   cmCathodeMainPnP2AxisZ.commandConfiguration.moveVelocity.velocity := 0.0;
   cmCathodeMainPnP2AxisZ.commandConfiguration.moveVelocity.acceleration := -1.0;
   cmCathodeMainPnP2AxisZ.commandConfiguration.moveVelocity.deceleration := -1.0;
   cmCathodeMainPnP2AxisZ.commandConfiguration.moveVelocity.jerk := -1.0;
   cmCathodeMainPnP2AxisZ.commandConfiguration.moveVelocity.direction := 0;
   cmCathodeMainPnP2AxisZ.commandConfiguration.moveVelocity.positionControlled := TRUE;
   cmCathodeMainPnP2AxisZ.commandConfiguration.moveVelocity.velocityChangeOnTheFly := FALSE;
   cmCathodeMainPnP2AxisZ.commandConfiguration.stop.deceleration := -1.0;
   cmCathodeMainPnP2AxisZ.commandConfiguration.stop.jerk := -1.0;
   cmCathodeMainPnP2AxisZ.commandConfiguration.stop.abortAcceleration := FALSE;
   cmCathodeMainPnP2AxisZ.commandConfiguration.fastStop.deceleration := -1.0;
   cmCathodeMainPnP2AxisZ.commandConfiguration.fastStop.jerk := -1.0;
   cmCathodeMainPnP2AxisZ.commandConfiguration.fastStop.abortAcceleration := FALSE;
   cmCathodeMainPnP2AxisZ.commandConfiguration.fastStop.replaceStopPossible := FALSE;
   cmCathodeMainPnP2AxisZ.commandConfiguration.torqueLimiting.limit := -1.0;
   cmCathodeMainPnP2AxisZ.commandConfiguration.torqueLimiting.mode := 0;
   cmCathodeMainPnP2AxisZ.commandConfiguration.homing.position := 0.0;
   cmCathodeMainPnP2AxisZ.commandConfiguration.homing.mode := 0;
   cmCathodeMainPnP2AxisZ.commandConfiguration.homing.sensor := 0;
   cmCathodeMainPnP2AxisZ.commandConfiguration.homing.extendedMode := -1;
   cmCathodeMainPnP2AxisZ.commandConfiguration.homing.extendedModeTorqueLimit := 0.0;
   cmCathodeMainPnP2AxisZ.commandConfiguration.homing.extendedModeTargetPosition := 0.0;
   cmCathodeMainPnP2AxisZ.commandConfiguration.posRelative.distance := 0.0;
   cmCathodeMainPnP2AxisZ.commandConfiguration.posRelative.velocity := -1.0;
   cmCathodeMainPnP2AxisZ.commandConfiguration.posRelative.acceleration := -1.0;
   cmCathodeMainPnP2AxisZ.commandConfiguration.posRelative.deceleration := -1.0;
   cmCathodeMainPnP2AxisZ.commandConfiguration.posRelative.jerk := -1.0;
   cmCathodeMainPnP2AxisZ.commandConfiguration.posRelative.direction := 0;
   cmCathodeMainPnP2AxisZ.commandConfiguration.posAbsolute.position := 0.0;
   cmCathodeMainPnP2AxisZ.commandConfiguration.posAbsolute.velocity := -1.0;
   cmCathodeMainPnP2AxisZ.commandConfiguration.posAbsolute.acceleration := -1.0;
   cmCathodeMainPnP2AxisZ.commandConfiguration.posAbsolute.deceleration := -1.0;
   cmCathodeMainPnP2AxisZ.commandConfiguration.posAbsolute.jerk := -1.0;
   cmCathodeMainPnP2AxisZ.commandConfiguration.posAbsolute.direction := 1;
   cmCathodeMainPnP2AxisZ.commandConfiguration.posAbsolute.positionChangeOnTheFly := FALSE;
   cmCathodeMainPnP2AxisZ.commandConfiguration.posAbsolute.velocityChangeOnTheFly := FALSE;
   cmCathodeMainPnP2AxisZ.commandConfiguration.posSuperimposed.distance := 0.0;
   cmCathodeMainPnP2AxisZ.commandConfiguration.posSuperimposed.velocityDiff := -1.0;
   cmCathodeMainPnP2AxisZ.commandConfiguration.posSuperimposed.acceleration := -1.0;
   cmCathodeMainPnP2AxisZ.commandConfiguration.posSuperimposed.deceleration := -1.0;
   cmCathodeMainPnP2AxisZ.commandConfiguration.posSuperimposed.jerk := -1.0;
   cmCathodeMainPnP2AxisZ.commandConfiguration.posSuperimposed.direction := 0;
   cmCathodeMainPnP2AxisZ.commandConfiguration.haltSuperimposed.deceleration := -1.0;
   cmCathodeMainPnP2AxisZ.commandConfiguration.haltSuperimposed.jerk := -1.0;
   cmCathodeMainPnP2AxisZ.commandConfiguration.haltSuperimposed.abortAcceleration := FALSE;
   cmCathodeMainPnP2AxisZ.commandConfiguration.gearInRelative.ratioNumerator := 1;
   cmCathodeMainPnP2AxisZ.commandConfiguration.gearInRelative.ratioDenominator := 1;
   cmCathodeMainPnP2AxisZ.commandConfiguration.gearInRelative.acceleration := -1.0;
   cmCathodeMainPnP2AxisZ.commandConfiguration.gearInRelative.deceleration := -1.0;
   cmCathodeMainPnP2AxisZ.commandConfiguration.gearInRelative.jerk := -1.0;
   cmCathodeMainPnP2AxisZ.commandConfiguration.gearInRelative.ratioChangeOnTheFly := FALSE;
   cmCathodeMainPnP2AxisZ.commandConfiguration.gearInAbsolute.ratioNumerator := 1;
   cmCathodeMainPnP2AxisZ.commandConfiguration.gearInAbsolute.ratioDenominator := 1;
   cmCathodeMainPnP2AxisZ.commandConfiguration.gearInAbsolute.masterSyncPosition := 0.0;
   cmCathodeMainPnP2AxisZ.commandConfiguration.gearInAbsolute.slaveSyncPosition := 0.0;
   cmCathodeMainPnP2AxisZ.commandConfiguration.gearInAbsolute.syncProfileReference := 1;
   cmCathodeMainPnP2AxisZ.commandConfiguration.gearInAbsolute.masterStartDistance := 0.0;
   cmCathodeMainPnP2AxisZ.commandConfiguration.gearInAbsolute.velocity := -1.0;
   cmCathodeMainPnP2AxisZ.commandConfiguration.gearInAbsolute.acceleration := -1.0;
   cmCathodeMainPnP2AxisZ.commandConfiguration.gearInAbsolute.deceleration := -1.0;
   cmCathodeMainPnP2AxisZ.commandConfiguration.gearInAbsolute.jerk := -1.0;
   cmCathodeMainPnP2AxisZ.commandConfiguration.gearInAbsolute.syncDirection := 1;
   cmCathodeMainPnP2AxisZ.commandConfiguration.gearInAbsolute.ratioChangeOnTheFly := FALSE;
   cmCathodeMainPnP2AxisZ.commandConfiguration.gearInVelocity.continuousUpdate := FALSE;
   cmCathodeMainPnP2AxisZ.commandConfiguration.gearInVelocity.ratioNumerator := 1;
   cmCathodeMainPnP2AxisZ.commandConfiguration.gearInVelocity.ratioDenominator := 1;
   cmCathodeMainPnP2AxisZ.commandConfiguration.gearInVelocity.acceleration := -1.0;
   cmCathodeMainPnP2AxisZ.commandConfiguration.gearInVelocity.deceleration := -1.0;
   cmCathodeMainPnP2AxisZ.commandConfiguration.gearInVelocity.jerk := -1.0;
   cmCathodeMainPnP2AxisZ.commandConfiguration.gearInVelocity.positionControlled := FALSE;
   cmCathodeMainPnP2AxisZ.commandConfiguration.camIn.masterOffset := 0.0;
   cmCathodeMainPnP2AxisZ.commandConfiguration.camIn.slaveOffset := 0.0;
   cmCathodeMainPnP2AxisZ.commandConfiguration.camIn.masterScaling := 1.0;
   cmCathodeMainPnP2AxisZ.commandConfiguration.camIn.slaveScaling := 1.0;
   cmCathodeMainPnP2AxisZ.commandConfiguration.camIn.masterSyncPosition := 0.0;
   cmCathodeMainPnP2AxisZ.commandConfiguration.camIn.syncProfileReference := 1;
   cmCathodeMainPnP2AxisZ.commandConfiguration.camIn.masterStartDistance := 0.0;
   cmCathodeMainPnP2AxisZ.commandConfiguration.camIn.velocity := -1.0;
   cmCathodeMainPnP2AxisZ.commandConfiguration.camIn.acceleration := -1.0;
   cmCathodeMainPnP2AxisZ.commandConfiguration.camIn.deceleration := -1.0;
   cmCathodeMainPnP2AxisZ.commandConfiguration.camIn.jerk := -1.0;
   cmCathodeMainPnP2AxisZ.commandConfiguration.camIn.applicationMode := 0;
   cmCathodeMainPnP2AxisZ.commandConfiguration.camIn.syncDirection := 1;
   cmCathodeMainPnP2AxisZ.commandConfiguration.gearOutCamOut.slavePosition := 0.0;
   cmCathodeMainPnP2AxisZ.commandConfiguration.gearOutCamOut.syncProfileReference := 1;
   cmCathodeMainPnP2AxisZ.commandConfiguration.gearOutCamOut.masterStopDistance := 0.0;
   cmCathodeMainPnP2AxisZ.commandConfiguration.gearOutCamOut.deceleration := -1.0;
   cmCathodeMainPnP2AxisZ.commandConfiguration.gearOutCamOut.jerk := -1.0;
   cmCathodeMainPnP2AxisZ.commandConfiguration.gearOutCamOut.syncOutDirection := 3;
   cmCathodeMainPnP2AxisZ.commandConfiguration.gearOutCamOut.gearOutCamOutMode := -1;
   cmCathodeMainPnP2AxisZ.commandConfiguration.phasing.phaseShift := 0.0;
   cmCathodeMainPnP2AxisZ.commandConfiguration.phasing.velocity := -1.0;
   cmCathodeMainPnP2AxisZ.commandConfiguration.phasing.acceleration := -1.0;
   cmCathodeMainPnP2AxisZ.commandConfiguration.phasing.deceleration := -1.0;
   cmCathodeMainPnP2AxisZ.commandConfiguration.phasing.jerk := -1.0;
   cmCathodeMainPnP2AxisZ.commandConfiguration.phasing.profileReference := 0;
   cmCathodeMainPnP2AxisZ.commandConfiguration.phasing.phasingDistance := 0.0;
   cmCathodeMainPnP2AxisZ.commandConfiguration.phasing.startPosition := 0.0;
   cmCathodeMainPnP2AxisZ.commandConfiguration.phasing.direction := 3;
   cmCathodeMainPnP2AxisZ.commandConfiguration.phasing.phaseAbsolute := TRUE;
   cmCathodeMainPnP2AxisZ.commandConfiguration.phasing.phaseShiftChangeOnTheFly := FALSE;
   cmCathodeMainPnP2AxisZ.commandConfiguration.offset.offset := 0.0;
   cmCathodeMainPnP2AxisZ.commandConfiguration.offset.profileReference := 1;
   cmCathodeMainPnP2AxisZ.commandConfiguration.offset.offsetDistance := 0.0;
   cmCathodeMainPnP2AxisZ.commandConfiguration.offset.startPosition := 0.0;
   cmCathodeMainPnP2AxisZ.commandConfiguration.offset.direction := 3;
   cmCathodeMainPnP2AxisZ.commandConfiguration.offset.offsetAbsolute := TRUE;
   cmCathodeMainPnP2AxisZ.commandConfiguration.offset.offsetChangeOnTheFly := FALSE;
   cmCathodeMainPnP2AxisZ.commands.enableAxis := FALSE;
   cmCathodeMainPnP2AxisZ.commands.resetAxis := FALSE;
   cmCathodeMainPnP2AxisZ.commands.openBrake := FALSE;
   cmCathodeMainPnP2AxisZ.commands.jogForward := FALSE;
   cmCathodeMainPnP2AxisZ.commands.jogBackward := FALSE;
   cmCathodeMainPnP2AxisZ.commands.moveVelocity := FALSE;
   cmCathodeMainPnP2AxisZ.commands.stop := FALSE;
   cmCathodeMainPnP2AxisZ.commands.fastStop := FALSE;
   cmCathodeMainPnP2AxisZ.commands.torqueLimiting := FALSE;
   cmCathodeMainPnP2AxisZ.commands.homing := FALSE;
   cmCathodeMainPnP2AxisZ.commands.posRelative := FALSE;
   cmCathodeMainPnP2AxisZ.commands.posAbsolute := FALSE;
   cmCathodeMainPnP2AxisZ.commands.posSuperimposed := FALSE;
   cmCathodeMainPnP2AxisZ.commands.haltSuperimposed := FALSE;
   cmCathodeMainPnP2AxisZ.commands.selectSetPosition := -1;
   cmCathodeMainPnP2AxisZ.commands.reset := FALSE;
   cmCathodeMainPnP2AxisZ.monitoring.valid := FALSE;
   cmCathodeMainPnP2AxisZ.monitoring.busy := TRUE;
   cmCathodeMainPnP2AxisZ.monitoring.error := TRUE;
   cmCathodeMainPnP2AxisZ.monitoring.status := 16#8600;
   cmCathodeMainPnP2AxisZ.monitoring.subfunctionStatus := 16#8001;
   cmCathodeMainPnP2AxisZ.monitoring.axisEnabled := FALSE;
   cmCathodeMainPnP2AxisZ.monitoring.resetActive := FALSE;
   cmCathodeMainPnP2AxisZ.monitoring.inVelocity := FALSE;
   cmCathodeMainPnP2AxisZ.monitoring.inLimitation := FALSE;
   cmCathodeMainPnP2AxisZ.monitoring.inClamping := FALSE;
   cmCathodeMainPnP2AxisZ.monitoring.startSync := FALSE;
   cmCathodeMainPnP2AxisZ.monitoring.inSync := FALSE;
   cmCathodeMainPnP2AxisZ.monitoring.inSimulation := FALSE;
   cmCathodeMainPnP2AxisZ.monitoring.jogSelected := FALSE;
   cmCathodeMainPnP2AxisZ.monitoring.moveVelocitySelected := FALSE;
   cmCathodeMainPnP2AxisZ.monitoring.stopSelected := FALSE;
   cmCathodeMainPnP2AxisZ.monitoring.fastStopSelected := FALSE;
   cmCathodeMainPnP2AxisZ.monitoring.torqueLimitingSelected := FALSE;
   cmCathodeMainPnP2AxisZ.monitoring.homingSelected := FALSE;
   cmCathodeMainPnP2AxisZ.monitoring.posRelativeSelected := FALSE;
   cmCathodeMainPnP2AxisZ.monitoring.posAbsoluteSelected := FALSE;
   cmCathodeMainPnP2AxisZ.monitoring.posSuperimposedSelected := FALSE;
   cmCathodeMainPnP2AxisZ.monitoring.haltSuperimposedSelected := FALSE;
   cmCathodeMainPnP2AxisZ.monitoring.commandBusy := FALSE;
   cmCathodeMainPnP2AxisZ.monitoring.commandDone := FALSE;
   cmCathodeMainPnP2AxisZ.monitoring.commandAborted := FALSE;
   cmCathodeMainPnP2AxisZ.monitoring.homingCommandBusy := FALSE;
   cmCathodeMainPnP2AxisZ.monitoring.homingCommandDone := FALSE;
   cmCathodeMainPnP2AxisZ.monitoring.homingCommandAborted := FALSE;
   cmCathodeMainPnP2AxisZ.monitoring.superimposedBusy := FALSE;
   cmCathodeMainPnP2AxisZ.monitoring.superimposedDone := FALSE;
   cmCathodeMainPnP2AxisZ.monitoring.superimposedAborted := FALSE;
   cmCathodeMainPnP2AxisZ.monitoring.actualPosition := 2.382;
   cmCathodeMainPnP2AxisZ.monitoring.actualSpeed := 0.0;
   cmCathodeMainPnP2AxisZ.monitoring.speedUnit := 1062;
   cmCathodeMainPnP2AxisZ.monitoring.positionUnit := 1013;
   cmCathodeMainPnP2AxisZ.monitoring.axisType := 1;
   cmCathodeMainPnP2AxisZ.monitoring.interlockGeneralOut := TRUE;
   cmCathodeMainPnP2AxisZ.monitoring.interlockJogForwardOut := TRUE;
   cmCathodeMainPnP2AxisZ.monitoring.interlockJogBackwardOut := TRUE;
   cmCathodeAlignTableAxisX.commandConfiguration.generalSettings.stopOnError := TRUE;
   cmCathodeAlignTableAxisX.commandConfiguration.generalSettings.resetWithRestart := FALSE;
   cmCathodeAlignTableAxisX.commandConfiguration.generalSettings.abortWaitingSyncCmd := TRUE;
   cmCathodeAlignTableAxisX.commandConfiguration.power.startMode := 1;
   cmCathodeAlignTableAxisX.commandConfiguration.power.stopMode := 0;
   cmCathodeAlignTableAxisX.commandConfiguration.power.syncMotionSimulation := FALSE;
   cmCathodeAlignTableAxisX.commandConfiguration.power.syncMotionSimulationExtendedMode := -1;
   cmCathodeAlignTableAxisX.commandConfiguration.jog.velocity := 0.0;
   cmCathodeAlignTableAxisX.commandConfiguration.jog.acceleration := -1.0;
   cmCathodeAlignTableAxisX.commandConfiguration.jog.deceleration := -1.0;
   cmCathodeAlignTableAxisX.commandConfiguration.jog.jerk := -1.0;
   cmCathodeAlignTableAxisX.commandConfiguration.jog.positionControlled := TRUE;
   cmCathodeAlignTableAxisX.commandConfiguration.jog.increment := 0.0;
   cmCathodeAlignTableAxisX.commandConfiguration.jog.mode := 0;
   cmCathodeAlignTableAxisX.commandConfiguration.moveVelocity.velocity := 0.0;
   cmCathodeAlignTableAxisX.commandConfiguration.moveVelocity.acceleration := -1.0;
   cmCathodeAlignTableAxisX.commandConfiguration.moveVelocity.deceleration := -1.0;
   cmCathodeAlignTableAxisX.commandConfiguration.moveVelocity.jerk := -1.0;
   cmCathodeAlignTableAxisX.commandConfiguration.moveVelocity.direction := 0;
   cmCathodeAlignTableAxisX.commandConfiguration.moveVelocity.positionControlled := TRUE;
   cmCathodeAlignTableAxisX.commandConfiguration.moveVelocity.velocityChangeOnTheFly := FALSE;
   cmCathodeAlignTableAxisX.commandConfiguration.stop.deceleration := -1.0;
   cmCathodeAlignTableAxisX.commandConfiguration.stop.jerk := -1.0;
   cmCathodeAlignTableAxisX.commandConfiguration.stop.abortAcceleration := FALSE;
   cmCathodeAlignTableAxisX.commandConfiguration.fastStop.deceleration := -1.0;
   cmCathodeAlignTableAxisX.commandConfiguration.fastStop.jerk := -1.0;
   cmCathodeAlignTableAxisX.commandConfiguration.fastStop.abortAcceleration := FALSE;
   cmCathodeAlignTableAxisX.commandConfiguration.fastStop.replaceStopPossible := FALSE;
   cmCathodeAlignTableAxisX.commandConfiguration.torqueLimiting.limit := -1.0;
   cmCathodeAlignTableAxisX.commandConfiguration.torqueLimiting.mode := 0;
   cmCathodeAlignTableAxisX.commandConfiguration.homing.position := 0.0;
   cmCathodeAlignTableAxisX.commandConfiguration.homing.mode := 0;
   cmCathodeAlignTableAxisX.commandConfiguration.homing.sensor := 0;
   cmCathodeAlignTableAxisX.commandConfiguration.homing.extendedMode := -1;
   cmCathodeAlignTableAxisX.commandConfiguration.homing.extendedModeTorqueLimit := 0.0;
   cmCathodeAlignTableAxisX.commandConfiguration.homing.extendedModeTargetPosition := 0.0;
   cmCathodeAlignTableAxisX.commandConfiguration.posRelative.distance := 0.0;
   cmCathodeAlignTableAxisX.commandConfiguration.posRelative.velocity := -1.0;
   cmCathodeAlignTableAxisX.commandConfiguration.posRelative.acceleration := -1.0;
   cmCathodeAlignTableAxisX.commandConfiguration.posRelative.deceleration := -1.0;
   cmCathodeAlignTableAxisX.commandConfiguration.posRelative.jerk := -1.0;
   cmCathodeAlignTableAxisX.commandConfiguration.posRelative.direction := 0;
   cmCathodeAlignTableAxisX.commandConfiguration.posAbsolute.position := 0.0;
   cmCathodeAlignTableAxisX.commandConfiguration.posAbsolute.velocity := -1.0;
   cmCathodeAlignTableAxisX.commandConfiguration.posAbsolute.acceleration := -1.0;
   cmCathodeAlignTableAxisX.commandConfiguration.posAbsolute.deceleration := -1.0;
   cmCathodeAlignTableAxisX.commandConfiguration.posAbsolute.jerk := -1.0;
   cmCathodeAlignTableAxisX.commandConfiguration.posAbsolute.direction := 1;
   cmCathodeAlignTableAxisX.commandConfiguration.posAbsolute.positionChangeOnTheFly := FALSE;
   cmCathodeAlignTableAxisX.commandConfiguration.posAbsolute.velocityChangeOnTheFly := FALSE;
   cmCathodeAlignTableAxisX.commandConfiguration.posSuperimposed.distance := 0.0;
   cmCathodeAlignTableAxisX.commandConfiguration.posSuperimposed.velocityDiff := -1.0;
   cmCathodeAlignTableAxisX.commandConfiguration.posSuperimposed.acceleration := -1.0;
   cmCathodeAlignTableAxisX.commandConfiguration.posSuperimposed.deceleration := -1.0;
   cmCathodeAlignTableAxisX.commandConfiguration.posSuperimposed.jerk := -1.0;
   cmCathodeAlignTableAxisX.commandConfiguration.posSuperimposed.direction := 0;
   cmCathodeAlignTableAxisX.commandConfiguration.haltSuperimposed.deceleration := -1.0;
   cmCathodeAlignTableAxisX.commandConfiguration.haltSuperimposed.jerk := -1.0;
   cmCathodeAlignTableAxisX.commandConfiguration.haltSuperimposed.abortAcceleration := FALSE;
   cmCathodeAlignTableAxisX.commandConfiguration.gearInRelative.ratioNumerator := 1;
   cmCathodeAlignTableAxisX.commandConfiguration.gearInRelative.ratioDenominator := 1;
   cmCathodeAlignTableAxisX.commandConfiguration.gearInRelative.acceleration := -1.0;
   cmCathodeAlignTableAxisX.commandConfiguration.gearInRelative.deceleration := -1.0;
   cmCathodeAlignTableAxisX.commandConfiguration.gearInRelative.jerk := -1.0;
   cmCathodeAlignTableAxisX.commandConfiguration.gearInRelative.ratioChangeOnTheFly := FALSE;
   cmCathodeAlignTableAxisX.commandConfiguration.gearInAbsolute.ratioNumerator := 1;
   cmCathodeAlignTableAxisX.commandConfiguration.gearInAbsolute.ratioDenominator := 1;
   cmCathodeAlignTableAxisX.commandConfiguration.gearInAbsolute.masterSyncPosition := 0.0;
   cmCathodeAlignTableAxisX.commandConfiguration.gearInAbsolute.slaveSyncPosition := 0.0;
   cmCathodeAlignTableAxisX.commandConfiguration.gearInAbsolute.syncProfileReference := 1;
   cmCathodeAlignTableAxisX.commandConfiguration.gearInAbsolute.masterStartDistance := 0.0;
   cmCathodeAlignTableAxisX.commandConfiguration.gearInAbsolute.velocity := -1.0;
   cmCathodeAlignTableAxisX.commandConfiguration.gearInAbsolute.acceleration := -1.0;
   cmCathodeAlignTableAxisX.commandConfiguration.gearInAbsolute.deceleration := -1.0;
   cmCathodeAlignTableAxisX.commandConfiguration.gearInAbsolute.jerk := -1.0;
   cmCathodeAlignTableAxisX.commandConfiguration.gearInAbsolute.syncDirection := 1;
   cmCathodeAlignTableAxisX.commandConfiguration.gearInAbsolute.ratioChangeOnTheFly := FALSE;
   cmCathodeAlignTableAxisX.commandConfiguration.gearInVelocity.continuousUpdate := FALSE;
   cmCathodeAlignTableAxisX.commandConfiguration.gearInVelocity.ratioNumerator := 1;
   cmCathodeAlignTableAxisX.commandConfiguration.gearInVelocity.ratioDenominator := 1;
   cmCathodeAlignTableAxisX.commandConfiguration.gearInVelocity.acceleration := -1.0;
   cmCathodeAlignTableAxisX.commandConfiguration.gearInVelocity.deceleration := -1.0;
   cmCathodeAlignTableAxisX.commandConfiguration.gearInVelocity.jerk := -1.0;
   cmCathodeAlignTableAxisX.commandConfiguration.gearInVelocity.positionControlled := FALSE;
   cmCathodeAlignTableAxisX.commandConfiguration.camIn.masterOffset := 0.0;
   cmCathodeAlignTableAxisX.commandConfiguration.camIn.slaveOffset := 0.0;
   cmCathodeAlignTableAxisX.commandConfiguration.camIn.masterScaling := 1.0;
   cmCathodeAlignTableAxisX.commandConfiguration.camIn.slaveScaling := 1.0;
   cmCathodeAlignTableAxisX.commandConfiguration.camIn.masterSyncPosition := 0.0;
   cmCathodeAlignTableAxisX.commandConfiguration.camIn.syncProfileReference := 1;
   cmCathodeAlignTableAxisX.commandConfiguration.camIn.masterStartDistance := 0.0;
   cmCathodeAlignTableAxisX.commandConfiguration.camIn.velocity := -1.0;
   cmCathodeAlignTableAxisX.commandConfiguration.camIn.acceleration := -1.0;
   cmCathodeAlignTableAxisX.commandConfiguration.camIn.deceleration := -1.0;
   cmCathodeAlignTableAxisX.commandConfiguration.camIn.jerk := -1.0;
   cmCathodeAlignTableAxisX.commandConfiguration.camIn.applicationMode := 0;
   cmCathodeAlignTableAxisX.commandConfiguration.camIn.syncDirection := 1;
   cmCathodeAlignTableAxisX.commandConfiguration.gearOutCamOut.slavePosition := 0.0;
   cmCathodeAlignTableAxisX.commandConfiguration.gearOutCamOut.syncProfileReference := 1;
   cmCathodeAlignTableAxisX.commandConfiguration.gearOutCamOut.masterStopDistance := 0.0;
   cmCathodeAlignTableAxisX.commandConfiguration.gearOutCamOut.deceleration := -1.0;
   cmCathodeAlignTableAxisX.commandConfiguration.gearOutCamOut.jerk := -1.0;
   cmCathodeAlignTableAxisX.commandConfiguration.gearOutCamOut.syncOutDirection := 3;
   cmCathodeAlignTableAxisX.commandConfiguration.gearOutCamOut.gearOutCamOutMode := -1;
   cmCathodeAlignTableAxisX.commandConfiguration.phasing.phaseShift := 0.0;
   cmCathodeAlignTableAxisX.commandConfiguration.phasing.velocity := -1.0;
   cmCathodeAlignTableAxisX.commandConfiguration.phasing.acceleration := -1.0;
   cmCathodeAlignTableAxisX.commandConfiguration.phasing.deceleration := -1.0;
   cmCathodeAlignTableAxisX.commandConfiguration.phasing.jerk := -1.0;
   cmCathodeAlignTableAxisX.commandConfiguration.phasing.profileReference := 0;
   cmCathodeAlignTableAxisX.commandConfiguration.phasing.phasingDistance := 0.0;
   cmCathodeAlignTableAxisX.commandConfiguration.phasing.startPosition := 0.0;
   cmCathodeAlignTableAxisX.commandConfiguration.phasing.direction := 3;
   cmCathodeAlignTableAxisX.commandConfiguration.phasing.phaseAbsolute := TRUE;
   cmCathodeAlignTableAxisX.commandConfiguration.phasing.phaseShiftChangeOnTheFly := FALSE;
   cmCathodeAlignTableAxisX.commandConfiguration.offset.offset := 0.0;
   cmCathodeAlignTableAxisX.commandConfiguration.offset.profileReference := 1;
   cmCathodeAlignTableAxisX.commandConfiguration.offset.offsetDistance := 0.0;
   cmCathodeAlignTableAxisX.commandConfiguration.offset.startPosition := 0.0;
   cmCathodeAlignTableAxisX.commandConfiguration.offset.direction := 3;
   cmCathodeAlignTableAxisX.commandConfiguration.offset.offsetAbsolute := TRUE;
   cmCathodeAlignTableAxisX.commandConfiguration.offset.offsetChangeOnTheFly := FALSE;
   cmCathodeAlignTableAxisX.commands.enableAxis := FALSE;
   cmCathodeAlignTableAxisX.commands.resetAxis := FALSE;
   cmCathodeAlignTableAxisX.commands.openBrake := FALSE;
   cmCathodeAlignTableAxisX.commands.jogForward := FALSE;
   cmCathodeAlignTableAxisX.commands.jogBackward := FALSE;
   cmCathodeAlignTableAxisX.commands.moveVelocity := FALSE;
   cmCathodeAlignTableAxisX.commands.stop := FALSE;
   cmCathodeAlignTableAxisX.commands.fastStop := FALSE;
   cmCathodeAlignTableAxisX.commands.torqueLimiting := FALSE;
   cmCathodeAlignTableAxisX.commands.homing := FALSE;
   cmCathodeAlignTableAxisX.commands.posRelative := FALSE;
   cmCathodeAlignTableAxisX.commands.posAbsolute := FALSE;
   cmCathodeAlignTableAxisX.commands.posSuperimposed := FALSE;
   cmCathodeAlignTableAxisX.commands.haltSuperimposed := FALSE;
   cmCathodeAlignTableAxisX.commands.selectSetPosition := -1;
   cmCathodeAlignTableAxisX.commands.reset := FALSE;
   cmCathodeAlignTableAxisX.monitoring.valid := FALSE;
   cmCathodeAlignTableAxisX.monitoring.busy := TRUE;
   cmCathodeAlignTableAxisX.monitoring.error := TRUE;
   cmCathodeAlignTableAxisX.monitoring.status := 16#8600;
   cmCathodeAlignTableAxisX.monitoring.subfunctionStatus := 16#8001;
   cmCathodeAlignTableAxisX.monitoring.axisEnabled := FALSE;
   cmCathodeAlignTableAxisX.monitoring.resetActive := FALSE;
   cmCathodeAlignTableAxisX.monitoring.inVelocity := FALSE;
   cmCathodeAlignTableAxisX.monitoring.inLimitation := FALSE;
   cmCathodeAlignTableAxisX.monitoring.inClamping := FALSE;
   cmCathodeAlignTableAxisX.monitoring.startSync := FALSE;
   cmCathodeAlignTableAxisX.monitoring.inSync := FALSE;
   cmCathodeAlignTableAxisX.monitoring.inSimulation := FALSE;
   cmCathodeAlignTableAxisX.monitoring.jogSelected := FALSE;
   cmCathodeAlignTableAxisX.monitoring.moveVelocitySelected := FALSE;
   cmCathodeAlignTableAxisX.monitoring.stopSelected := FALSE;
   cmCathodeAlignTableAxisX.monitoring.fastStopSelected := FALSE;
   cmCathodeAlignTableAxisX.monitoring.torqueLimitingSelected := FALSE;
   cmCathodeAlignTableAxisX.monitoring.homingSelected := FALSE;
   cmCathodeAlignTableAxisX.monitoring.posRelativeSelected := FALSE;
   cmCathodeAlignTableAxisX.monitoring.posAbsoluteSelected := FALSE;
   cmCathodeAlignTableAxisX.monitoring.posSuperimposedSelected := FALSE;
   cmCathodeAlignTableAxisX.monitoring.haltSuperimposedSelected := FALSE;
   cmCathodeAlignTableAxisX.monitoring.commandBusy := FALSE;
   cmCathodeAlignTableAxisX.monitoring.commandDone := FALSE;
   cmCathodeAlignTableAxisX.monitoring.commandAborted := FALSE;
   cmCathodeAlignTableAxisX.monitoring.homingCommandBusy := FALSE;
   cmCathodeAlignTableAxisX.monitoring.homingCommandDone := FALSE;
   cmCathodeAlignTableAxisX.monitoring.homingCommandAborted := FALSE;
   cmCathodeAlignTableAxisX.monitoring.superimposedBusy := FALSE;
   cmCathodeAlignTableAxisX.monitoring.superimposedDone := FALSE;
   cmCathodeAlignTableAxisX.monitoring.superimposedAborted := FALSE;
   cmCathodeAlignTableAxisX.monitoring.actualPosition := -0.929;
   cmCathodeAlignTableAxisX.monitoring.actualSpeed := 0.0;
   cmCathodeAlignTableAxisX.monitoring.speedUnit := 1062;
   cmCathodeAlignTableAxisX.monitoring.positionUnit := 1013;
   cmCathodeAlignTableAxisX.monitoring.axisType := 1;
   cmCathodeAlignTableAxisX.monitoring.interlockGeneralOut := TRUE;
   cmCathodeAlignTableAxisX.monitoring.interlockJogForwardOut := TRUE;
   cmCathodeAlignTableAxisX.monitoring.interlockJogBackwardOut := TRUE;
   cmCathodeAlignTableAxisY1.commandConfiguration.generalSettings.stopOnError := TRUE;
   cmCathodeAlignTableAxisY1.commandConfiguration.generalSettings.resetWithRestart := FALSE;
   cmCathodeAlignTableAxisY1.commandConfiguration.generalSettings.abortWaitingSyncCmd := TRUE;
   cmCathodeAlignTableAxisY1.commandConfiguration.power.startMode := 1;
   cmCathodeAlignTableAxisY1.commandConfiguration.power.stopMode := 0;
   cmCathodeAlignTableAxisY1.commandConfiguration.power.syncMotionSimulation := FALSE;
   cmCathodeAlignTableAxisY1.commandConfiguration.power.syncMotionSimulationExtendedMode := -1;
   cmCathodeAlignTableAxisY1.commandConfiguration.jog.velocity := 0.0;
   cmCathodeAlignTableAxisY1.commandConfiguration.jog.acceleration := -1.0;
   cmCathodeAlignTableAxisY1.commandConfiguration.jog.deceleration := -1.0;
   cmCathodeAlignTableAxisY1.commandConfiguration.jog.jerk := -1.0;
   cmCathodeAlignTableAxisY1.commandConfiguration.jog.positionControlled := TRUE;
   cmCathodeAlignTableAxisY1.commandConfiguration.jog.increment := 0.0;
   cmCathodeAlignTableAxisY1.commandConfiguration.jog.mode := 0;
   cmCathodeAlignTableAxisY1.commandConfiguration.moveVelocity.velocity := 0.0;
   cmCathodeAlignTableAxisY1.commandConfiguration.moveVelocity.acceleration := -1.0;
   cmCathodeAlignTableAxisY1.commandConfiguration.moveVelocity.deceleration := -1.0;
   cmCathodeAlignTableAxisY1.commandConfiguration.moveVelocity.jerk := -1.0;
   cmCathodeAlignTableAxisY1.commandConfiguration.moveVelocity.direction := 0;
   cmCathodeAlignTableAxisY1.commandConfiguration.moveVelocity.positionControlled := TRUE;
   cmCathodeAlignTableAxisY1.commandConfiguration.moveVelocity.velocityChangeOnTheFly := FALSE;
   cmCathodeAlignTableAxisY1.commandConfiguration.stop.deceleration := -1.0;
   cmCathodeAlignTableAxisY1.commandConfiguration.stop.jerk := -1.0;
   cmCathodeAlignTableAxisY1.commandConfiguration.stop.abortAcceleration := FALSE;
   cmCathodeAlignTableAxisY1.commandConfiguration.fastStop.deceleration := -1.0;
   cmCathodeAlignTableAxisY1.commandConfiguration.fastStop.jerk := -1.0;
   cmCathodeAlignTableAxisY1.commandConfiguration.fastStop.abortAcceleration := FALSE;
   cmCathodeAlignTableAxisY1.commandConfiguration.fastStop.replaceStopPossible := FALSE;
   cmCathodeAlignTableAxisY1.commandConfiguration.torqueLimiting.limit := -1.0;
   cmCathodeAlignTableAxisY1.commandConfiguration.torqueLimiting.mode := 0;
   cmCathodeAlignTableAxisY1.commandConfiguration.homing.position := 0.0;
   cmCathodeAlignTableAxisY1.commandConfiguration.homing.mode := 0;
   cmCathodeAlignTableAxisY1.commandConfiguration.homing.sensor := 0;
   cmCathodeAlignTableAxisY1.commandConfiguration.homing.extendedMode := -1;
   cmCathodeAlignTableAxisY1.commandConfiguration.homing.extendedModeTorqueLimit := 0.0;
   cmCathodeAlignTableAxisY1.commandConfiguration.homing.extendedModeTargetPosition := 0.0;
   cmCathodeAlignTableAxisY1.commandConfiguration.posRelative.distance := 0.0;
   cmCathodeAlignTableAxisY1.commandConfiguration.posRelative.velocity := -1.0;
   cmCathodeAlignTableAxisY1.commandConfiguration.posRelative.acceleration := -1.0;
   cmCathodeAlignTableAxisY1.commandConfiguration.posRelative.deceleration := -1.0;
   cmCathodeAlignTableAxisY1.commandConfiguration.posRelative.jerk := -1.0;
   cmCathodeAlignTableAxisY1.commandConfiguration.posRelative.direction := 0;
   cmCathodeAlignTableAxisY1.commandConfiguration.posAbsolute.position := 0.0;
   cmCathodeAlignTableAxisY1.commandConfiguration.posAbsolute.velocity := -1.0;
   cmCathodeAlignTableAxisY1.commandConfiguration.posAbsolute.acceleration := -1.0;
   cmCathodeAlignTableAxisY1.commandConfiguration.posAbsolute.deceleration := -1.0;
   cmCathodeAlignTableAxisY1.commandConfiguration.posAbsolute.jerk := -1.0;
   cmCathodeAlignTableAxisY1.commandConfiguration.posAbsolute.direction := 1;
   cmCathodeAlignTableAxisY1.commandConfiguration.posAbsolute.positionChangeOnTheFly := FALSE;
   cmCathodeAlignTableAxisY1.commandConfiguration.posAbsolute.velocityChangeOnTheFly := FALSE;
   cmCathodeAlignTableAxisY1.commandConfiguration.posSuperimposed.distance := 0.0;
   cmCathodeAlignTableAxisY1.commandConfiguration.posSuperimposed.velocityDiff := -1.0;
   cmCathodeAlignTableAxisY1.commandConfiguration.posSuperimposed.acceleration := -1.0;
   cmCathodeAlignTableAxisY1.commandConfiguration.posSuperimposed.deceleration := -1.0;
   cmCathodeAlignTableAxisY1.commandConfiguration.posSuperimposed.jerk := -1.0;
   cmCathodeAlignTableAxisY1.commandConfiguration.posSuperimposed.direction := 0;
   cmCathodeAlignTableAxisY1.commandConfiguration.haltSuperimposed.deceleration := -1.0;
   cmCathodeAlignTableAxisY1.commandConfiguration.haltSuperimposed.jerk := -1.0;
   cmCathodeAlignTableAxisY1.commandConfiguration.haltSuperimposed.abortAcceleration := FALSE;
   cmCathodeAlignTableAxisY1.commandConfiguration.gearInRelative.ratioNumerator := 1;
   cmCathodeAlignTableAxisY1.commandConfiguration.gearInRelative.ratioDenominator := 1;
   cmCathodeAlignTableAxisY1.commandConfiguration.gearInRelative.acceleration := -1.0;
   cmCathodeAlignTableAxisY1.commandConfiguration.gearInRelative.deceleration := -1.0;
   cmCathodeAlignTableAxisY1.commandConfiguration.gearInRelative.jerk := -1.0;
   cmCathodeAlignTableAxisY1.commandConfiguration.gearInRelative.ratioChangeOnTheFly := FALSE;
   cmCathodeAlignTableAxisY1.commandConfiguration.gearInAbsolute.ratioNumerator := 1;
   cmCathodeAlignTableAxisY1.commandConfiguration.gearInAbsolute.ratioDenominator := 1;
   cmCathodeAlignTableAxisY1.commandConfiguration.gearInAbsolute.masterSyncPosition := 0.0;
   cmCathodeAlignTableAxisY1.commandConfiguration.gearInAbsolute.slaveSyncPosition := 0.0;
   cmCathodeAlignTableAxisY1.commandConfiguration.gearInAbsolute.syncProfileReference := 1;
   cmCathodeAlignTableAxisY1.commandConfiguration.gearInAbsolute.masterStartDistance := 0.0;
   cmCathodeAlignTableAxisY1.commandConfiguration.gearInAbsolute.velocity := -1.0;
   cmCathodeAlignTableAxisY1.commandConfiguration.gearInAbsolute.acceleration := -1.0;
   cmCathodeAlignTableAxisY1.commandConfiguration.gearInAbsolute.deceleration := -1.0;
   cmCathodeAlignTableAxisY1.commandConfiguration.gearInAbsolute.jerk := -1.0;
   cmCathodeAlignTableAxisY1.commandConfiguration.gearInAbsolute.syncDirection := 1;
   cmCathodeAlignTableAxisY1.commandConfiguration.gearInAbsolute.ratioChangeOnTheFly := FALSE;
   cmCathodeAlignTableAxisY1.commandConfiguration.gearInVelocity.continuousUpdate := FALSE;
   cmCathodeAlignTableAxisY1.commandConfiguration.gearInVelocity.ratioNumerator := 1;
   cmCathodeAlignTableAxisY1.commandConfiguration.gearInVelocity.ratioDenominator := 1;
   cmCathodeAlignTableAxisY1.commandConfiguration.gearInVelocity.acceleration := -1.0;
   cmCathodeAlignTableAxisY1.commandConfiguration.gearInVelocity.deceleration := -1.0;
   cmCathodeAlignTableAxisY1.commandConfiguration.gearInVelocity.jerk := -1.0;
   cmCathodeAlignTableAxisY1.commandConfiguration.gearInVelocity.positionControlled := FALSE;
   cmCathodeAlignTableAxisY1.commandConfiguration.camIn.masterOffset := 0.0;
   cmCathodeAlignTableAxisY1.commandConfiguration.camIn.slaveOffset := 0.0;
   cmCathodeAlignTableAxisY1.commandConfiguration.camIn.masterScaling := 1.0;
   cmCathodeAlignTableAxisY1.commandConfiguration.camIn.slaveScaling := 1.0;
   cmCathodeAlignTableAxisY1.commandConfiguration.camIn.masterSyncPosition := 0.0;
   cmCathodeAlignTableAxisY1.commandConfiguration.camIn.syncProfileReference := 1;
   cmCathodeAlignTableAxisY1.commandConfiguration.camIn.masterStartDistance := 0.0;
   cmCathodeAlignTableAxisY1.commandConfiguration.camIn.velocity := -1.0;
   cmCathodeAlignTableAxisY1.commandConfiguration.camIn.acceleration := -1.0;
   cmCathodeAlignTableAxisY1.commandConfiguration.camIn.deceleration := -1.0;
   cmCathodeAlignTableAxisY1.commandConfiguration.camIn.jerk := -1.0;
   cmCathodeAlignTableAxisY1.commandConfiguration.camIn.applicationMode := 0;
   cmCathodeAlignTableAxisY1.commandConfiguration.camIn.syncDirection := 1;
   cmCathodeAlignTableAxisY1.commandConfiguration.gearOutCamOut.slavePosition := 0.0;
   cmCathodeAlignTableAxisY1.commandConfiguration.gearOutCamOut.syncProfileReference := 1;
   cmCathodeAlignTableAxisY1.commandConfiguration.gearOutCamOut.masterStopDistance := 0.0;
   cmCathodeAlignTableAxisY1.commandConfiguration.gearOutCamOut.deceleration := -1.0;
   cmCathodeAlignTableAxisY1.commandConfiguration.gearOutCamOut.jerk := -1.0;
   cmCathodeAlignTableAxisY1.commandConfiguration.gearOutCamOut.syncOutDirection := 3;
   cmCathodeAlignTableAxisY1.commandConfiguration.gearOutCamOut.gearOutCamOutMode := -1;
   cmCathodeAlignTableAxisY1.commandConfiguration.phasing.phaseShift := 0.0;
   cmCathodeAlignTableAxisY1.commandConfiguration.phasing.velocity := -1.0;
   cmCathodeAlignTableAxisY1.commandConfiguration.phasing.acceleration := -1.0;
   cmCathodeAlignTableAxisY1.commandConfiguration.phasing.deceleration := -1.0;
   cmCathodeAlignTableAxisY1.commandConfiguration.phasing.jerk := -1.0;
   cmCathodeAlignTableAxisY1.commandConfiguration.phasing.profileReference := 0;
   cmCathodeAlignTableAxisY1.commandConfiguration.phasing.phasingDistance := 0.0;
   cmCathodeAlignTableAxisY1.commandConfiguration.phasing.startPosition := 0.0;
   cmCathodeAlignTableAxisY1.commandConfiguration.phasing.direction := 3;
   cmCathodeAlignTableAxisY1.commandConfiguration.phasing.phaseAbsolute := TRUE;
   cmCathodeAlignTableAxisY1.commandConfiguration.phasing.phaseShiftChangeOnTheFly := FALSE;
   cmCathodeAlignTableAxisY1.commandConfiguration.offset.offset := 0.0;
   cmCathodeAlignTableAxisY1.commandConfiguration.offset.profileReference := 1;
   cmCathodeAlignTableAxisY1.commandConfiguration.offset.offsetDistance := 0.0;
   cmCathodeAlignTableAxisY1.commandConfiguration.offset.startPosition := 0.0;
   cmCathodeAlignTableAxisY1.commandConfiguration.offset.direction := 3;
   cmCathodeAlignTableAxisY1.commandConfiguration.offset.offsetAbsolute := TRUE;
   cmCathodeAlignTableAxisY1.commandConfiguration.offset.offsetChangeOnTheFly := FALSE;
   cmCathodeAlignTableAxisY1.commands.enableAxis := FALSE;
   cmCathodeAlignTableAxisY1.commands.resetAxis := FALSE;
   cmCathodeAlignTableAxisY1.commands.openBrake := FALSE;
   cmCathodeAlignTableAxisY1.commands.jogForward := FALSE;
   cmCathodeAlignTableAxisY1.commands.jogBackward := FALSE;
   cmCathodeAlignTableAxisY1.commands.moveVelocity := FALSE;
   cmCathodeAlignTableAxisY1.commands.stop := FALSE;
   cmCathodeAlignTableAxisY1.commands.fastStop := FALSE;
   cmCathodeAlignTableAxisY1.commands.torqueLimiting := FALSE;
   cmCathodeAlignTableAxisY1.commands.homing := FALSE;
   cmCathodeAlignTableAxisY1.commands.posRelative := FALSE;
   cmCathodeAlignTableAxisY1.commands.posAbsolute := FALSE;
   cmCathodeAlignTableAxisY1.commands.posSuperimposed := FALSE;
   cmCathodeAlignTableAxisY1.commands.haltSuperimposed := FALSE;
   cmCathodeAlignTableAxisY1.commands.selectSetPosition := -1;
   cmCathodeAlignTableAxisY1.commands.reset := FALSE;
   cmCathodeAlignTableAxisY1.monitoring.valid := FALSE;
   cmCathodeAlignTableAxisY1.monitoring.busy := TRUE;
   cmCathodeAlignTableAxisY1.monitoring.error := TRUE;
   cmCathodeAlignTableAxisY1.monitoring.status := 16#8600;
   cmCathodeAlignTableAxisY1.monitoring.subfunctionStatus := 16#8001;
   cmCathodeAlignTableAxisY1.monitoring.axisEnabled := FALSE;
   cmCathodeAlignTableAxisY1.monitoring.resetActive := FALSE;
   cmCathodeAlignTableAxisY1.monitoring.inVelocity := FALSE;
   cmCathodeAlignTableAxisY1.monitoring.inLimitation := FALSE;
   cmCathodeAlignTableAxisY1.monitoring.inClamping := FALSE;
   cmCathodeAlignTableAxisY1.monitoring.startSync := FALSE;
   cmCathodeAlignTableAxisY1.monitoring.inSync := FALSE;
   cmCathodeAlignTableAxisY1.monitoring.inSimulation := FALSE;
   cmCathodeAlignTableAxisY1.monitoring.jogSelected := FALSE;
   cmCathodeAlignTableAxisY1.monitoring.moveVelocitySelected := FALSE;
   cmCathodeAlignTableAxisY1.monitoring.stopSelected := FALSE;
   cmCathodeAlignTableAxisY1.monitoring.fastStopSelected := FALSE;
   cmCathodeAlignTableAxisY1.monitoring.torqueLimitingSelected := FALSE;
   cmCathodeAlignTableAxisY1.monitoring.homingSelected := FALSE;
   cmCathodeAlignTableAxisY1.monitoring.posRelativeSelected := FALSE;
   cmCathodeAlignTableAxisY1.monitoring.posAbsoluteSelected := FALSE;
   cmCathodeAlignTableAxisY1.monitoring.posSuperimposedSelected := FALSE;
   cmCathodeAlignTableAxisY1.monitoring.haltSuperimposedSelected := FALSE;
   cmCathodeAlignTableAxisY1.monitoring.commandBusy := FALSE;
   cmCathodeAlignTableAxisY1.monitoring.commandDone := FALSE;
   cmCathodeAlignTableAxisY1.monitoring.commandAborted := FALSE;
   cmCathodeAlignTableAxisY1.monitoring.homingCommandBusy := FALSE;
   cmCathodeAlignTableAxisY1.monitoring.homingCommandDone := FALSE;
   cmCathodeAlignTableAxisY1.monitoring.homingCommandAborted := FALSE;
   cmCathodeAlignTableAxisY1.monitoring.superimposedBusy := FALSE;
   cmCathodeAlignTableAxisY1.monitoring.superimposedDone := FALSE;
   cmCathodeAlignTableAxisY1.monitoring.superimposedAborted := FALSE;
   cmCathodeAlignTableAxisY1.monitoring.actualPosition := 0.15;
   cmCathodeAlignTableAxisY1.monitoring.actualSpeed := 0.0;
   cmCathodeAlignTableAxisY1.monitoring.speedUnit := 1062;
   cmCathodeAlignTableAxisY1.monitoring.positionUnit := 1013;
   cmCathodeAlignTableAxisY1.monitoring.axisType := 1;
   cmCathodeAlignTableAxisY1.monitoring.interlockGeneralOut := TRUE;
   cmCathodeAlignTableAxisY1.monitoring.interlockJogForwardOut := TRUE;
   cmCathodeAlignTableAxisY1.monitoring.interlockJogBackwardOut := TRUE;
   cmCathodeAlignTableAxisY2.commandConfiguration.generalSettings.stopOnError := TRUE;
   cmCathodeAlignTableAxisY2.commandConfiguration.generalSettings.resetWithRestart := FALSE;
   cmCathodeAlignTableAxisY2.commandConfiguration.generalSettings.abortWaitingSyncCmd := TRUE;
   cmCathodeAlignTableAxisY2.commandConfiguration.power.startMode := 1;
   cmCathodeAlignTableAxisY2.commandConfiguration.power.stopMode := 0;
   cmCathodeAlignTableAxisY2.commandConfiguration.power.syncMotionSimulation := FALSE;
   cmCathodeAlignTableAxisY2.commandConfiguration.power.syncMotionSimulationExtendedMode := -1;
   cmCathodeAlignTableAxisY2.commandConfiguration.jog.velocity := 0.0;
   cmCathodeAlignTableAxisY2.commandConfiguration.jog.acceleration := -1.0;
   cmCathodeAlignTableAxisY2.commandConfiguration.jog.deceleration := -1.0;
   cmCathodeAlignTableAxisY2.commandConfiguration.jog.jerk := -1.0;
   cmCathodeAlignTableAxisY2.commandConfiguration.jog.positionControlled := TRUE;
   cmCathodeAlignTableAxisY2.commandConfiguration.jog.increment := 0.0;
   cmCathodeAlignTableAxisY2.commandConfiguration.jog.mode := 0;
   cmCathodeAlignTableAxisY2.commandConfiguration.moveVelocity.velocity := 0.0;
   cmCathodeAlignTableAxisY2.commandConfiguration.moveVelocity.acceleration := -1.0;
   cmCathodeAlignTableAxisY2.commandConfiguration.moveVelocity.deceleration := -1.0;
   cmCathodeAlignTableAxisY2.commandConfiguration.moveVelocity.jerk := -1.0;
   cmCathodeAlignTableAxisY2.commandConfiguration.moveVelocity.direction := 0;
   cmCathodeAlignTableAxisY2.commandConfiguration.moveVelocity.positionControlled := TRUE;
   cmCathodeAlignTableAxisY2.commandConfiguration.moveVelocity.velocityChangeOnTheFly := FALSE;
   cmCathodeAlignTableAxisY2.commandConfiguration.stop.deceleration := -1.0;
   cmCathodeAlignTableAxisY2.commandConfiguration.stop.jerk := -1.0;
   cmCathodeAlignTableAxisY2.commandConfiguration.stop.abortAcceleration := FALSE;
   cmCathodeAlignTableAxisY2.commandConfiguration.fastStop.deceleration := -1.0;
   cmCathodeAlignTableAxisY2.commandConfiguration.fastStop.jerk := -1.0;
   cmCathodeAlignTableAxisY2.commandConfiguration.fastStop.abortAcceleration := FALSE;
   cmCathodeAlignTableAxisY2.commandConfiguration.fastStop.replaceStopPossible := FALSE;
   cmCathodeAlignTableAxisY2.commandConfiguration.torqueLimiting.limit := -1.0;
   cmCathodeAlignTableAxisY2.commandConfiguration.torqueLimiting.mode := 0;
   cmCathodeAlignTableAxisY2.commandConfiguration.homing.position := 0.0;
   cmCathodeAlignTableAxisY2.commandConfiguration.homing.mode := 0;
   cmCathodeAlignTableAxisY2.commandConfiguration.homing.sensor := 0;
   cmCathodeAlignTableAxisY2.commandConfiguration.homing.extendedMode := -1;
   cmCathodeAlignTableAxisY2.commandConfiguration.homing.extendedModeTorqueLimit := 0.0;
   cmCathodeAlignTableAxisY2.commandConfiguration.homing.extendedModeTargetPosition := 0.0;
   cmCathodeAlignTableAxisY2.commandConfiguration.posRelative.distance := 0.0;
   cmCathodeAlignTableAxisY2.commandConfiguration.posRelative.velocity := -1.0;
   cmCathodeAlignTableAxisY2.commandConfiguration.posRelative.acceleration := -1.0;
   cmCathodeAlignTableAxisY2.commandConfiguration.posRelative.deceleration := -1.0;
   cmCathodeAlignTableAxisY2.commandConfiguration.posRelative.jerk := -1.0;
   cmCathodeAlignTableAxisY2.commandConfiguration.posRelative.direction := 0;
   cmCathodeAlignTableAxisY2.commandConfiguration.posAbsolute.position := 0.0;
   cmCathodeAlignTableAxisY2.commandConfiguration.posAbsolute.velocity := -1.0;
   cmCathodeAlignTableAxisY2.commandConfiguration.posAbsolute.acceleration := -1.0;
   cmCathodeAlignTableAxisY2.commandConfiguration.posAbsolute.deceleration := -1.0;
   cmCathodeAlignTableAxisY2.commandConfiguration.posAbsolute.jerk := -1.0;
   cmCathodeAlignTableAxisY2.commandConfiguration.posAbsolute.direction := 1;
   cmCathodeAlignTableAxisY2.commandConfiguration.posAbsolute.positionChangeOnTheFly := FALSE;
   cmCathodeAlignTableAxisY2.commandConfiguration.posAbsolute.velocityChangeOnTheFly := FALSE;
   cmCathodeAlignTableAxisY2.commandConfiguration.posSuperimposed.distance := 0.0;
   cmCathodeAlignTableAxisY2.commandConfiguration.posSuperimposed.velocityDiff := -1.0;
   cmCathodeAlignTableAxisY2.commandConfiguration.posSuperimposed.acceleration := -1.0;
   cmCathodeAlignTableAxisY2.commandConfiguration.posSuperimposed.deceleration := -1.0;
   cmCathodeAlignTableAxisY2.commandConfiguration.posSuperimposed.jerk := -1.0;
   cmCathodeAlignTableAxisY2.commandConfiguration.posSuperimposed.direction := 0;
   cmCathodeAlignTableAxisY2.commandConfiguration.haltSuperimposed.deceleration := -1.0;
   cmCathodeAlignTableAxisY2.commandConfiguration.haltSuperimposed.jerk := -1.0;
   cmCathodeAlignTableAxisY2.commandConfiguration.haltSuperimposed.abortAcceleration := FALSE;
   cmCathodeAlignTableAxisY2.commandConfiguration.gearInRelative.ratioNumerator := 1;
   cmCathodeAlignTableAxisY2.commandConfiguration.gearInRelative.ratioDenominator := 1;
   cmCathodeAlignTableAxisY2.commandConfiguration.gearInRelative.acceleration := -1.0;
   cmCathodeAlignTableAxisY2.commandConfiguration.gearInRelative.deceleration := -1.0;
   cmCathodeAlignTableAxisY2.commandConfiguration.gearInRelative.jerk := -1.0;
   cmCathodeAlignTableAxisY2.commandConfiguration.gearInRelative.ratioChangeOnTheFly := FALSE;
   cmCathodeAlignTableAxisY2.commandConfiguration.gearInAbsolute.ratioNumerator := 1;
   cmCathodeAlignTableAxisY2.commandConfiguration.gearInAbsolute.ratioDenominator := 1;
   cmCathodeAlignTableAxisY2.commandConfiguration.gearInAbsolute.masterSyncPosition := 0.0;
   cmCathodeAlignTableAxisY2.commandConfiguration.gearInAbsolute.slaveSyncPosition := 0.0;
   cmCathodeAlignTableAxisY2.commandConfiguration.gearInAbsolute.syncProfileReference := 1;
   cmCathodeAlignTableAxisY2.commandConfiguration.gearInAbsolute.masterStartDistance := 0.0;
   cmCathodeAlignTableAxisY2.commandConfiguration.gearInAbsolute.velocity := -1.0;
   cmCathodeAlignTableAxisY2.commandConfiguration.gearInAbsolute.acceleration := -1.0;
   cmCathodeAlignTableAxisY2.commandConfiguration.gearInAbsolute.deceleration := -1.0;
   cmCathodeAlignTableAxisY2.commandConfiguration.gearInAbsolute.jerk := -1.0;
   cmCathodeAlignTableAxisY2.commandConfiguration.gearInAbsolute.syncDirection := 1;
   cmCathodeAlignTableAxisY2.commandConfiguration.gearInAbsolute.ratioChangeOnTheFly := FALSE;
   cmCathodeAlignTableAxisY2.commandConfiguration.gearInVelocity.continuousUpdate := FALSE;
   cmCathodeAlignTableAxisY2.commandConfiguration.gearInVelocity.ratioNumerator := 1;
   cmCathodeAlignTableAxisY2.commandConfiguration.gearInVelocity.ratioDenominator := 1;
   cmCathodeAlignTableAxisY2.commandConfiguration.gearInVelocity.acceleration := -1.0;
   cmCathodeAlignTableAxisY2.commandConfiguration.gearInVelocity.deceleration := -1.0;
   cmCathodeAlignTableAxisY2.commandConfiguration.gearInVelocity.jerk := -1.0;
   cmCathodeAlignTableAxisY2.commandConfiguration.gearInVelocity.positionControlled := FALSE;
   cmCathodeAlignTableAxisY2.commandConfiguration.camIn.masterOffset := 0.0;
   cmCathodeAlignTableAxisY2.commandConfiguration.camIn.slaveOffset := 0.0;
   cmCathodeAlignTableAxisY2.commandConfiguration.camIn.masterScaling := 1.0;
   cmCathodeAlignTableAxisY2.commandConfiguration.camIn.slaveScaling := 1.0;
   cmCathodeAlignTableAxisY2.commandConfiguration.camIn.masterSyncPosition := 0.0;
   cmCathodeAlignTableAxisY2.commandConfiguration.camIn.syncProfileReference := 1;
   cmCathodeAlignTableAxisY2.commandConfiguration.camIn.masterStartDistance := 0.0;
   cmCathodeAlignTableAxisY2.commandConfiguration.camIn.velocity := -1.0;
   cmCathodeAlignTableAxisY2.commandConfiguration.camIn.acceleration := -1.0;
   cmCathodeAlignTableAxisY2.commandConfiguration.camIn.deceleration := -1.0;
   cmCathodeAlignTableAxisY2.commandConfiguration.camIn.jerk := -1.0;
   cmCathodeAlignTableAxisY2.commandConfiguration.camIn.applicationMode := 0;
   cmCathodeAlignTableAxisY2.commandConfiguration.camIn.syncDirection := 1;
   cmCathodeAlignTableAxisY2.commandConfiguration.gearOutCamOut.slavePosition := 0.0;
   cmCathodeAlignTableAxisY2.commandConfiguration.gearOutCamOut.syncProfileReference := 1;
   cmCathodeAlignTableAxisY2.commandConfiguration.gearOutCamOut.masterStopDistance := 0.0;
   cmCathodeAlignTableAxisY2.commandConfiguration.gearOutCamOut.deceleration := -1.0;
   cmCathodeAlignTableAxisY2.commandConfiguration.gearOutCamOut.jerk := -1.0;
   cmCathodeAlignTableAxisY2.commandConfiguration.gearOutCamOut.syncOutDirection := 3;
   cmCathodeAlignTableAxisY2.commandConfiguration.gearOutCamOut.gearOutCamOutMode := -1;
   cmCathodeAlignTableAxisY2.commandConfiguration.phasing.phaseShift := 0.0;
   cmCathodeAlignTableAxisY2.commandConfiguration.phasing.velocity := -1.0;
   cmCathodeAlignTableAxisY2.commandConfiguration.phasing.acceleration := -1.0;
   cmCathodeAlignTableAxisY2.commandConfiguration.phasing.deceleration := -1.0;
   cmCathodeAlignTableAxisY2.commandConfiguration.phasing.jerk := -1.0;
   cmCathodeAlignTableAxisY2.commandConfiguration.phasing.profileReference := 0;
   cmCathodeAlignTableAxisY2.commandConfiguration.phasing.phasingDistance := 0.0;
   cmCathodeAlignTableAxisY2.commandConfiguration.phasing.startPosition := 0.0;
   cmCathodeAlignTableAxisY2.commandConfiguration.phasing.direction := 3;
   cmCathodeAlignTableAxisY2.commandConfiguration.phasing.phaseAbsolute := TRUE;
   cmCathodeAlignTableAxisY2.commandConfiguration.phasing.phaseShiftChangeOnTheFly := FALSE;
   cmCathodeAlignTableAxisY2.commandConfiguration.offset.offset := 0.0;
   cmCathodeAlignTableAxisY2.commandConfiguration.offset.profileReference := 1;
   cmCathodeAlignTableAxisY2.commandConfiguration.offset.offsetDistance := 0.0;
   cmCathodeAlignTableAxisY2.commandConfiguration.offset.startPosition := 0.0;
   cmCathodeAlignTableAxisY2.commandConfiguration.offset.direction := 3;
   cmCathodeAlignTableAxisY2.commandConfiguration.offset.offsetAbsolute := TRUE;
   cmCathodeAlignTableAxisY2.commandConfiguration.offset.offsetChangeOnTheFly := FALSE;
   cmCathodeAlignTableAxisY2.commands.enableAxis := FALSE;
   cmCathodeAlignTableAxisY2.commands.resetAxis := FALSE;
   cmCathodeAlignTableAxisY2.commands.openBrake := FALSE;
   cmCathodeAlignTableAxisY2.commands.jogForward := FALSE;
   cmCathodeAlignTableAxisY2.commands.jogBackward := FALSE;
   cmCathodeAlignTableAxisY2.commands.moveVelocity := FALSE;
   cmCathodeAlignTableAxisY2.commands.stop := FALSE;
   cmCathodeAlignTableAxisY2.commands.fastStop := FALSE;
   cmCathodeAlignTableAxisY2.commands.torqueLimiting := FALSE;
   cmCathodeAlignTableAxisY2.commands.homing := FALSE;
   cmCathodeAlignTableAxisY2.commands.posRelative := FALSE;
   cmCathodeAlignTableAxisY2.commands.posAbsolute := FALSE;
   cmCathodeAlignTableAxisY2.commands.posSuperimposed := FALSE;
   cmCathodeAlignTableAxisY2.commands.haltSuperimposed := FALSE;
   cmCathodeAlignTableAxisY2.commands.selectSetPosition := -1;
   cmCathodeAlignTableAxisY2.commands.reset := FALSE;
   cmCathodeAlignTableAxisY2.monitoring.valid := FALSE;
   cmCathodeAlignTableAxisY2.monitoring.busy := TRUE;
   cmCathodeAlignTableAxisY2.monitoring.error := TRUE;
   cmCathodeAlignTableAxisY2.monitoring.status := 16#8600;
   cmCathodeAlignTableAxisY2.monitoring.subfunctionStatus := 16#8001;
   cmCathodeAlignTableAxisY2.monitoring.axisEnabled := FALSE;
   cmCathodeAlignTableAxisY2.monitoring.resetActive := FALSE;
   cmCathodeAlignTableAxisY2.monitoring.inVelocity := FALSE;
   cmCathodeAlignTableAxisY2.monitoring.inLimitation := FALSE;
   cmCathodeAlignTableAxisY2.monitoring.inClamping := FALSE;
   cmCathodeAlignTableAxisY2.monitoring.startSync := FALSE;
   cmCathodeAlignTableAxisY2.monitoring.inSync := FALSE;
   cmCathodeAlignTableAxisY2.monitoring.inSimulation := FALSE;
   cmCathodeAlignTableAxisY2.monitoring.jogSelected := FALSE;
   cmCathodeAlignTableAxisY2.monitoring.moveVelocitySelected := FALSE;
   cmCathodeAlignTableAxisY2.monitoring.stopSelected := FALSE;
   cmCathodeAlignTableAxisY2.monitoring.fastStopSelected := FALSE;
   cmCathodeAlignTableAxisY2.monitoring.torqueLimitingSelected := FALSE;
   cmCathodeAlignTableAxisY2.monitoring.homingSelected := FALSE;
   cmCathodeAlignTableAxisY2.monitoring.posRelativeSelected := FALSE;
   cmCathodeAlignTableAxisY2.monitoring.posAbsoluteSelected := FALSE;
   cmCathodeAlignTableAxisY2.monitoring.posSuperimposedSelected := FALSE;
   cmCathodeAlignTableAxisY2.monitoring.haltSuperimposedSelected := FALSE;
   cmCathodeAlignTableAxisY2.monitoring.commandBusy := FALSE;
   cmCathodeAlignTableAxisY2.monitoring.commandDone := FALSE;
   cmCathodeAlignTableAxisY2.monitoring.commandAborted := FALSE;
   cmCathodeAlignTableAxisY2.monitoring.homingCommandBusy := FALSE;
   cmCathodeAlignTableAxisY2.monitoring.homingCommandDone := FALSE;
   cmCathodeAlignTableAxisY2.monitoring.homingCommandAborted := FALSE;
   cmCathodeAlignTableAxisY2.monitoring.superimposedBusy := FALSE;
   cmCathodeAlignTableAxisY2.monitoring.superimposedDone := FALSE;
   cmCathodeAlignTableAxisY2.monitoring.superimposedAborted := FALSE;
   cmCathodeAlignTableAxisY2.monitoring.actualPosition := -0.959;
   cmCathodeAlignTableAxisY2.monitoring.actualSpeed := 0.0;
   cmCathodeAlignTableAxisY2.monitoring.speedUnit := 1062;
   cmCathodeAlignTableAxisY2.monitoring.positionUnit := 1013;
   cmCathodeAlignTableAxisY2.monitoring.axisType := 1;
   cmCathodeAlignTableAxisY2.monitoring.interlockGeneralOut := TRUE;
   cmCathodeAlignTableAxisY2.monitoring.interlockJogForwardOut := TRUE;
   cmCathodeAlignTableAxisY2.monitoring.interlockJogBackwardOut := TRUE;
   cmCathodeMainPnP1SuctionPlateVacuum.commands.commandHomePos := FALSE;
   cmCathodeMainPnP1SuctionPlateVacuum.commands.commandWorkPos := FALSE;
   cmCathodeMainPnP1SuctionPlateVacuum.commands.reset := FALSE;
   cmCathodeMainPnP1SuctionPlateVacuum.monitoring.valid := TRUE;
   cmCathodeMainPnP1SuctionPlateVacuum.monitoring.busy := TRUE;
   cmCathodeMainPnP1SuctionPlateVacuum.monitoring.error := FALSE;
   cmCathodeMainPnP1SuctionPlateVacuum.monitoring.status := 16#7003;
   cmCathodeMainPnP1SuctionPlateVacuum.monitoring.inHomePos := TRUE;
   cmCathodeMainPnP1SuctionPlateVacuum.monitoring.inWorkPos := FALSE;
   cmCathodeMainPnP1SuctionPlateVacuum.monitoring.interlockWorkPosOut := TRUE;
   cmCathodeMainPnP1SuctionPlateVacuum.monitoring.interlockHomePosOut := TRUE;
   cmCathodeMainPnP2SuctionPlateVacuum.commands.commandHomePos := FALSE;
   cmCathodeMainPnP2SuctionPlateVacuum.commands.commandWorkPos := FALSE;
   cmCathodeMainPnP2SuctionPlateVacuum.commands.reset := FALSE;
   cmCathodeMainPnP2SuctionPlateVacuum.monitoring.valid := TRUE;
   cmCathodeMainPnP2SuctionPlateVacuum.monitoring.busy := TRUE;
   cmCathodeMainPnP2SuctionPlateVacuum.monitoring.error := FALSE;
   cmCathodeMainPnP2SuctionPlateVacuum.monitoring.status := 16#7003;
   cmCathodeMainPnP2SuctionPlateVacuum.monitoring.inHomePos := TRUE;
   cmCathodeMainPnP2SuctionPlateVacuum.monitoring.inWorkPos := FALSE;
   cmCathodeMainPnP2SuctionPlateVacuum.monitoring.interlockWorkPosOut := TRUE;
   cmCathodeMainPnP2SuctionPlateVacuum.monitoring.interlockHomePosOut := TRUE;
   cmCathodeAlignTableSuctionPlateVacuum.commands.commandHomePos := FALSE;
   cmCathodeAlignTableSuctionPlateVacuum.commands.commandWorkPos := FALSE;
   cmCathodeAlignTableSuctionPlateVacuum.commands.reset := FALSE;
   cmCathodeAlignTableSuctionPlateVacuum.monitoring.valid := TRUE;
   cmCathodeAlignTableSuctionPlateVacuum.monitoring.busy := TRUE;
   cmCathodeAlignTableSuctionPlateVacuum.monitoring.error := FALSE;
   cmCathodeAlignTableSuctionPlateVacuum.monitoring.status := 16#7003;
   cmCathodeAlignTableSuctionPlateVacuum.monitoring.inHomePos := TRUE;
   cmCathodeAlignTableSuctionPlateVacuum.monitoring.inWorkPos := FALSE;
   cmCathodeAlignTableSuctionPlateVacuum.monitoring.interlockWorkPosOut := TRUE;
   cmCathodeAlignTableSuctionPlateVacuum.monitoring.interlockHomePosOut := TRUE;
   cmCathodeGlassCleaning.commands.commandHomePos := FALSE;
   cmCathodeGlassCleaning.commands.commandWorkPos := FALSE;
   cmCathodeGlassCleaning.commands.reset := FALSE;
   cmCathodeGlassCleaning.monitoring.valid := TRUE;
   cmCathodeGlassCleaning.monitoring.busy := TRUE;
   cmCathodeGlassCleaning.monitoring.error := FALSE;
   cmCathodeGlassCleaning.monitoring.status := 16#7003;
   cmCathodeGlassCleaning.monitoring.inHomePos := FALSE;
   cmCathodeGlassCleaning.monitoring.inWorkPos := FALSE;
   cmCathodeGlassCleaning.monitoring.interlockWorkPosOut := TRUE;
   cmCathodeGlassCleaning.monitoring.interlockHomePosOut := TRUE;
   cmCathodeNgPnpUpDown.commands.commandHomePos := FALSE;
   cmCathodeNgPnpUpDown.commands.commandWorkPos := FALSE;
   cmCathodeNgPnpUpDown.commands.reset := FALSE;
   cmCathodeNgPnp1stFwdBwd.commands.commandHomePos := FALSE;
   cmCathodeNgPnp1stFwdBwd.commands.commandWorkPos := FALSE;
   cmCathodeNgPnp1stFwdBwd.commands.reset := FALSE;
   cmCathodeNgPnp2ndFwdBwd.commands.commandHomePos := FALSE;
   cmCathodeNgPnp2ndFwdBwd.commands.commandWorkPos := FALSE;
   cmCathodeNgPnp2ndFwdBwd.commands.reset := FALSE;
   cmCathodeMaintenanceMovingFixFwdBwd.commands.commandHomePos := FALSE;
   cmCathodeMaintenanceMovingFixFwdBwd.commands.commandWorkPos := FALSE;
   cmCathodeMaintenanceMovingFixFwdBwd.commands.reset := FALSE;
   cmCathodeMaintenanceMovingFixFwdBwd.monitoring.valid := TRUE;
   cmCathodeMaintenanceMovingFixFwdBwd.monitoring.busy := TRUE;
   cmCathodeMaintenanceMovingFixFwdBwd.monitoring.error := FALSE;
   cmCathodeMaintenanceMovingFixFwdBwd.monitoring.status := 16#7003;
   cmCathodeMaintenanceMovingFixFwdBwd.monitoring.inHomePos := FALSE;
   cmCathodeMaintenanceMovingFixFwdBwd.monitoring.inWorkPos := TRUE;
   cmCathodeMaintenanceMovingFixFwdBwd.monitoring.interlockWorkPosOut := TRUE;
   cmCathodeMaintenanceMovingFixFwdBwd.monitoring.interlockHomePosOut := TRUE;
   cmCathodeNgBoxLiftUpDown.commands.commandHomePos := FALSE;
   cmCathodeNgBoxLiftUpDown.commands.commandWorkPos := FALSE;
   cmCathodeNgBoxLiftUpDown.commands.reset := FALSE;
   cmCathodeNgBoxLiftUpDown.monitoring.valid := TRUE;
   cmCathodeNgBoxLiftUpDown.monitoring.busy := TRUE;
   cmCathodeNgBoxLiftUpDown.monitoring.error := FALSE;
   cmCathodeNgBoxLiftUpDown.monitoring.status := 16#7101;
   cmCathodeNgBoxLiftUpDown.monitoring.inHomePos := TRUE;
   cmCathodeNgBoxLiftUpDown.monitoring.inWorkPos := FALSE;
   cmCathodeNgBoxLiftUpDown.monitoring.interlockWorkPosOut := FALSE;
   cmCathodeNgBoxLiftUpDown.monitoring.interlockHomePosOut := TRUE;
   cmCathodeNgBoxLockUpDown.commands.commandHomePos := FALSE;
   cmCathodeNgBoxLockUpDown.commands.commandWorkPos := FALSE;
   cmCathodeNgBoxLockUpDown.commands.reset := FALSE;
   cmCathodeNgBoxLockUpDown.monitoring.valid := TRUE;
   cmCathodeNgBoxLockUpDown.monitoring.busy := TRUE;
   cmCathodeNgBoxLockUpDown.monitoring.error := FALSE;
   cmCathodeNgBoxLockUpDown.monitoring.status := 16#7003;
   cmCathodeNgBoxLockUpDown.monitoring.inHomePos := TRUE;
   cmCathodeNgBoxLockUpDown.monitoring.inWorkPos := FALSE;
   cmCathodeNgBoxLockUpDown.monitoring.interlockWorkPosOut := TRUE;
   cmCathodeNgBoxLockUpDown.monitoring.interlockHomePosOut := TRUE;
   cmCathodeNgPnpVaccum.commands.commandHomePos := FALSE;
   cmCathodeNgPnpVaccum.commands.commandWorkPos := FALSE;
   cmCathodeNgPnpVaccum.commands.reset := FALSE;
   cmCathodeNgPnpVaccum.monitoring.valid := TRUE;
   cmCathodeNgPnpVaccum.monitoring.busy := TRUE;
   cmCathodeNgPnpVaccum.monitoring.error := FALSE;
   cmCathodeNgPnpVaccum.monitoring.status := 16#7003;
   cmCathodeNgPnpVaccum.monitoring.inHomePos := TRUE;
   cmCathodeNgPnpVaccum.monitoring.inWorkPos := FALSE;
   cmCathodeNgPnpVaccum.monitoring.interlockWorkPosOut := TRUE;
   cmCathodeNgPnpVaccum.monitoring.interlockHomePosOut := TRUE;
   cmCathodeConveyorCoverFwdBwd.commands.commandHomePos := FALSE;
   cmCathodeConveyorCoverFwdBwd.commands.commandWorkPos := FALSE;
   cmCathodeConveyorCoverFwdBwd.commands.reset := FALSE;
   cmCathodeConveyorCoverFwdBwd.monitoring.valid := TRUE;
   cmCathodeConveyorCoverFwdBwd.monitoring.busy := TRUE;
   cmCathodeConveyorCoverFwdBwd.monitoring.error := FALSE;
   cmCathodeConveyorCoverFwdBwd.monitoring.status := 16#7003;
   cmCathodeConveyorCoverFwdBwd.monitoring.inHomePos := FALSE;
   cmCathodeConveyorCoverFwdBwd.monitoring.inWorkPos := FALSE;
   cmCathodeConveyorCoverFwdBwd.monitoring.interlockWorkPosOut := TRUE;
   cmCathodeConveyorCoverFwdBwd.monitoring.interlockHomePosOut := TRUE;
   cmCathodeConveyorPickUpBlower.commands.commandHomePos := FALSE;
   cmCathodeConveyorPickUpBlower.commands.commandWorkPos := FALSE;
   cmCathodeConveyorPickUpBlower.commands.reset := FALSE;
   cmCathodeConveyorPickUpBlower.monitoring.valid := TRUE;
   cmCathodeConveyorPickUpBlower.monitoring.busy := TRUE;
   cmCathodeConveyorPickUpBlower.monitoring.error := FALSE;
   cmCathodeConveyorPickUpBlower.monitoring.status := 16#7003;
   cmCathodeConveyorPickUpBlower.monitoring.inHomePos := FALSE;
   cmCathodeConveyorPickUpBlower.monitoring.inWorkPos := FALSE;
   cmCathodeConveyorPickUpBlower.monitoring.interlockWorkPosOut := TRUE;
   cmCathodeConveyorPickUpBlower.monitoring.interlockHomePosOut := TRUE;
END_DATA_BLOCK
